FUNCTION F_ResetTimersAndRCPTimes : BOOL
VAR_IN_OUT // These are references to the actual TON instances and the RCP structure
    fbPause_TON : TON;
    fbRamp_TON  : FB_TON_Pausable;
    fbHold_TON  : FB_TON_Pausable;
END_VAR

// Reset the timers by setting IN to FALSE
fbPause_TON(IN:=FALSE); // Calling the TON FB instances
fbRamp_TON(IN:=FALSE, Pause:=FALSE);
fbHold_TON(IN:=FALSE, Pause:=FALSE);

// Reset the elapsed times in the RCP structure
RCP.Pause_ET := T#0S;
RCP.RecipeRunET.ET := T#0S;
RCP.RecipeRunET.Mode := E_RecipeRunETMode.None;

F_ResetTimersAndRCPTimes := TRUE; // Indicate successful execution (optional)

END_FUNCTION

(* stored: Version 1.1.0.1, ProductVersion 3.1.4026.11
   POU F_ResetTimersAndRCPTimes: Id {cad1d9c5-016c-4366-ba0d-91e43630a276}, SpecialFunc None *)
